FUNCTION_BLOCK SPLIT_AL_INTO_AB (* this Function splits the 8 AB (BYTE) adapters from a AL (LWORD) *)
  (* Standard: 61499-2; Description: Copyright (c) 2026 Meisterschulen am Ostbahnhof SPDX-License-Identifier: EPL-2.0 *)
  (* Version 1.0, 2026-05-16, Franz Höpfinger, Meisterschulen am Ostbahnhof, initial API and implementation and/or initial documentation *)
  PACKAGE adapter::splitting;
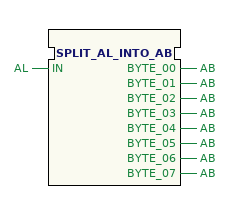
  SOCKETS
    IN : adapter::types::unidirectional::AL; (* LWORD Input *)
  END_SOCKETS
  PLUGS
    BYTE_00 : adapter::types::unidirectional::AB; (* Byte 0 *)
    BYTE_01 : adapter::types::unidirectional::AB; (* Byte 1 *)
    BYTE_02 : adapter::types::unidirectional::AB; (* Byte 2 *)
    BYTE_03 : adapter::types::unidirectional::AB; (* Byte 3 *)
    BYTE_04 : adapter::types::unidirectional::AB; (* Byte 4 *)
    BYTE_05 : adapter::types::unidirectional::AB; (* Byte 5 *)
    BYTE_06 : adapter::types::unidirectional::AB; (* Byte 6 *)
    BYTE_07 : adapter::types::unidirectional::AB; (* Byte 7 *)
  END_PLUGS
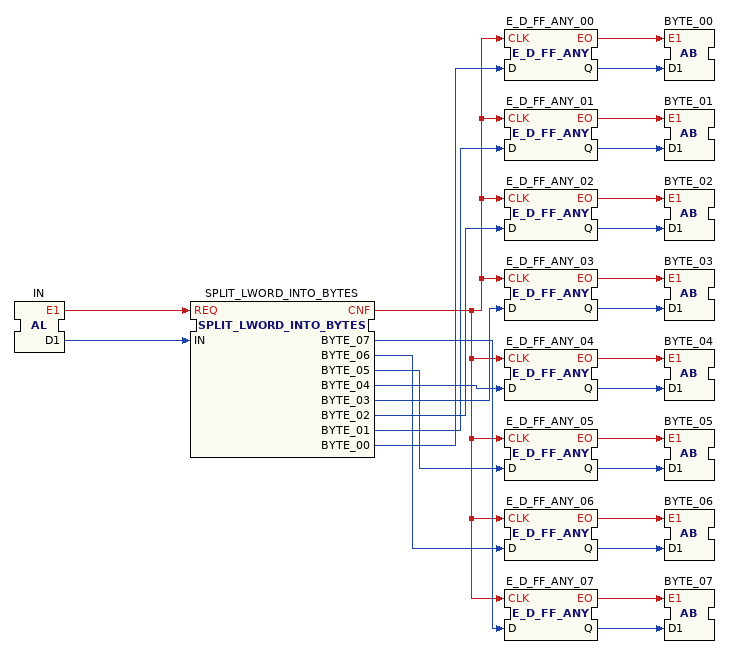
  FBS
    E_D_FF_ANY_00 : iec61499::events::E_D_FF_ANY;
    E_D_FF_ANY_01 : iec61499::events::E_D_FF_ANY;
    E_D_FF_ANY_02 : iec61499::events::E_D_FF_ANY;
    E_D_FF_ANY_03 : iec61499::events::E_D_FF_ANY;
    E_D_FF_ANY_04 : iec61499::events::E_D_FF_ANY;
    E_D_FF_ANY_05 : iec61499::events::E_D_FF_ANY;
    E_D_FF_ANY_06 : iec61499::events::E_D_FF_ANY;
    E_D_FF_ANY_07 : iec61499::events::E_D_FF_ANY;
    SPLIT_LWORD_INTO_BYTES : eclipse4diac::utils::splitting::SPLIT_LWORD_INTO_BYTES;
  END_FBS
  EVENT_CONNECTIONS
    IN.E1 TO SPLIT_LWORD_INTO_BYTES.REQ;
    SPLIT_LWORD_INTO_BYTES.CNF TO E_D_FF_ANY_00.CLK;
    SPLIT_LWORD_INTO_BYTES.CNF TO E_D_FF_ANY_01.CLK;
    SPLIT_LWORD_INTO_BYTES.CNF TO E_D_FF_ANY_02.CLK;
    SPLIT_LWORD_INTO_BYTES.CNF TO E_D_FF_ANY_03.CLK;
    SPLIT_LWORD_INTO_BYTES.CNF TO E_D_FF_ANY_04.CLK;
    SPLIT_LWORD_INTO_BYTES.CNF TO E_D_FF_ANY_05.CLK;
    SPLIT_LWORD_INTO_BYTES.CNF TO E_D_FF_ANY_06.CLK;
    SPLIT_LWORD_INTO_BYTES.CNF TO E_D_FF_ANY_07.CLK;
    E_D_FF_ANY_00.EO TO BYTE_00.E1;
    E_D_FF_ANY_01.EO TO BYTE_01.E1;
    E_D_FF_ANY_02.EO TO BYTE_02.E1;
    E_D_FF_ANY_03.EO TO BYTE_03.E1;
    E_D_FF_ANY_04.EO TO BYTE_04.E1;
    E_D_FF_ANY_05.EO TO BYTE_05.E1;
    E_D_FF_ANY_06.EO TO BYTE_06.E1;
    E_D_FF_ANY_07.EO TO BYTE_07.E1;
  END_CONNECTIONS
  DATA_CONNECTIONS
    IN.D1 TO SPLIT_LWORD_INTO_BYTES.IN;
    SPLIT_LWORD_INTO_BYTES.BYTE_07 TO E_D_FF_ANY_07.D;
    SPLIT_LWORD_INTO_BYTES.BYTE_06 TO E_D_FF_ANY_06.D;
    SPLIT_LWORD_INTO_BYTES.BYTE_05 TO E_D_FF_ANY_05.D;
    SPLIT_LWORD_INTO_BYTES.BYTE_04 TO E_D_FF_ANY_04.D;
    SPLIT_LWORD_INTO_BYTES.BYTE_03 TO E_D_FF_ANY_03.D;
    SPLIT_LWORD_INTO_BYTES.BYTE_02 TO E_D_FF_ANY_02.D;
    SPLIT_LWORD_INTO_BYTES.BYTE_01 TO E_D_FF_ANY_01.D;
    SPLIT_LWORD_INTO_BYTES.BYTE_00 TO E_D_FF_ANY_00.D;
    E_D_FF_ANY_00.Q TO BYTE_00.D1;
    E_D_FF_ANY_01.Q TO BYTE_01.D1;
    E_D_FF_ANY_02.Q TO BYTE_02.D1;
    E_D_FF_ANY_03.Q TO BYTE_03.D1;
    E_D_FF_ANY_04.Q TO BYTE_04.D1;
    E_D_FF_ANY_05.Q TO BYTE_05.D1;
    E_D_FF_ANY_06.Q TO BYTE_06.D1;
    E_D_FF_ANY_07.Q TO BYTE_07.D1;
  END_CONNECTIONS
END_FUNCTION_BLOCK
